{attribute 'linkalways'} 
{attribute 'no_explicit_call' := 'This FB is a CLASS and must be accessed using methods or properties'}
{attribute 'enable_dynamic_creation'}
FUNCTION_BLOCK _ETcVnFilterDirection EXTENDS EnumDatatypeBase
VAR
	localData : ETcVnFilterDirection;
	activeData : REFERENCE TO ETcVnFilterDirection;
	enumBaseDatatype : _INT(localData);
END_VAR

METHOD PRIVATE AddLocalEnumeration
VAR_INPUT
	Enumeration : T_MAXSTRING;
	Value : ETcVnFilterDirection;
END_VAR
AddEnumeration(Enumeration, Value);
END_METHOD

PROPERTY PUBLIC Address : PVOID
GET
Address := ADR(activeData);
END_GET
END_PROPERTY

METHOD PUBLIC ClearReference
VAR_INPUT
END_VAR
activeData REF= localData;
SetBaseDatatypeReference();
END_METHOD

METHOD PUBLIC Clone : I_Datatype
VAR
    pClone : POINTER TO _ETcVnFilterDirection;
END_VAR
pClone := __NEW(_ETcVnFilterDirection(InitialValue := Value));
Clone := pClone^;
END_METHOD

METHOD FB_init : BOOL
VAR_INPUT
	bInitRetains : BOOL; // if TRUE, the retain variables are initialized (warm start / cold start)
	bInCopyCode : BOOL;  // if TRUE, the instance afterwards gets moved into the copy code (online change)
	InitialValue : ETcVnFilterDirection;
END_VAR
localData := InitialValue;
AddBaseDatatype(enumBaseDatatype);
ClearReference();

AddLocalEnumeration('TCVN_FD_X', ETcVnFilterDirection.TCVN_FD_X);
AddLocalEnumeration('TCVN_FD_Y', ETcVnFilterDirection.TCVN_FD_Y);
END_METHOD

PROPERTY PUBLIC Identifier : T_MAXSTRING
GET
Identifier := 'ETcVnFilterDirection';
END_GET
END_PROPERTY

METHOD IsEnumeratorValueEqual : BOOL
VAR_INPUT
	Enumerator : I_KeyValueForwardEnumerator;
END_VAR
VAR
	storedValue : ETcVnFilterDirection;
END_VAR
IF NOT Enumerator.TryGet(storedValue) THEN
	RETURN;
END_IF

IsEnumeratorValueEqual := storedValue = activeData;
END_METHOD

METHOD PUBLIC MakeReferenceTo
VAR_INPUT
	ReferenceTarget : REFERENCE TO ETcVnFilterDirection;
END_VAR
activeData REF= ReferenceTarget;
SetBaseDatatypeReference();
END_METHOD

METHOD PROTECTED SetBaseDatatypeReference
VAR_INPUT
END_VAR
enumBaseDatatype.MakeReferenceTo(activeData);
END_METHOD

PROPERTY PUBLIC Size : UDINT
GET
Size := SIZEOF(activeData);
END_GET
END_PROPERTY

METHOD TryMakeReferenceTo : BOOL
VAR_INPUT
	Target : I_Datatype;
END_VAR
VAR
	targetAsEnum : I_EnumDatatype;
	pTargetData : POINTER TO ETcVnFilterDirection;
END_VAR
IF NOT Target.TryResolveAsEnumDatatype(targetAsEnum) THEN
	RETURN;
END_IF

IF targetAsEnum.Identifier <> Identifier THEN
	RETURN;
END_IF

pTargetData := Target.Address;
activeData REF= pTargetData^;
SetBaseDatatypeReference();
TryMakeReferenceTo := TRUE;
END_METHOD

PROPERTY PUBLIC Value : ETcVnFilterDirection
GET
Value := activeData;
END_GET
SET
activeData := Value;
END_SET
END_PROPERTY

END_FUNCTION_BLOCK

(* stored: Version 1.1.0.1, ProductVersion 3.1.4024.13
   POU _ETcVnFilterDirection: Id {9bea03f5-9610-0af9-3da1-a622a79edc4b}, SpecialFunc None
   Folder Core: Id {2e7f368d-630d-08ac-0197-bb04a00e207f}
   Folder Protected: Id {21ead6ba-95c0-029d-3ba3-fdb77d98af83}
   Folder Customize: Id {763fa483-3376-0f54-29ea-7be3c9689015}
   Folder Constructor: Id {ff3c39af-286b-07fe-1675-83029097ba0b}
   Folder Private: Id {e34ee56f-6594-0e2f-390c-102f441cb978}
   Folder Protected: Id {f34e3029-1626-0e21-3ad9-4c65559350fd}
   Method AddLocalEnumeration: Id {20f9fa4e-57cb-0af4-22f4-94f2b87b6ae9}
   Property Address: Id {16de46f7-0257-0852-2552-345d2a149cbc}
   Get Get: Id {1830c61e-8230-0788-29c2-eebf8cf3b0f4}
   Method ClearReference: Id {bf37ab42-96f9-06de-2305-9006e427f549}
   Method Clone: Id {384b6513-1b04-0f6e-04bc-0708046cca34}
   Method FB_init: Id {49215c61-0902-0948-2913-d6ad288a395e}
   Property Identifier: Id {67e68f79-91b8-0816-3811-eec47d1aae85}
   Get Get: Id {385409b5-3c0d-0b7c-0d3d-23afd511e618}
   Method IsEnumeratorValueEqual: Id {6df1c1fd-bc38-0cb1-379c-0bcf93b8c842}
   Method MakeReferenceTo: Id {e8ae3af0-226b-02fb-202b-12b8243481a7}
   Method SetBaseDatatypeReference: Id {9b327cdd-687a-045a-04c0-388f26270312}
   Property Size: Id {af987f68-4bb2-0352-29f6-37dc704d09cd}
   Get Get: Id {3ef8241e-7c0c-08ce-3f4f-3dd04b88f7dd}
   Method TryMakeReferenceTo: Id {988c2079-2b94-03d2-2c40-49ff5d4c0ae8}
   Property Value: Id {c18e112a-d2bf-0f8a-0177-5accfaad7994}
   Get Get: Id {deffb621-e0d9-085a-2fe1-e5556a9e90bf}
   Set Set: Id {8ca8de34-d422-084b-2893-92ae3820f780} *)
